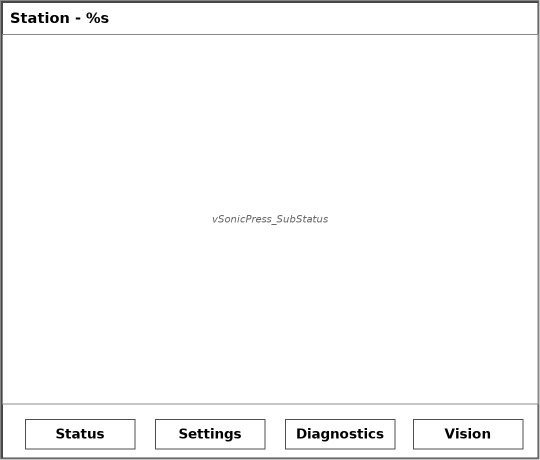
VISUALIZATION vSonicPress_Main  // 540x460
VAR_IN_OUT
	fbMachine: fbSonicPress;
	fbPIM: fbPIM_Station_V3;
	stTestParams:stSonicPress_TestParams;
END_VAR
    Rectangle (1,1 538x458)
    Rectangle (285,419 110x30), "Diagnostics"
        OnMouseClick: FrameSelectionChange Selection=SelectedFrame=57fd262e-2fea-4fde-aa72-b89d7183eaaf, Selection=2, GlobSel=AssignType=Expression, SelType=Locally
        OnMouseClick: execute { fbMachine.bTestMode:= FALSE; }
    Rectangle (155,419 110x30), "Settings"
        OnMouseClick: FrameSelectionChange Selection=SelectedFrame=57fd262e-2fea-4fde-aa72-b89d7183eaaf, Selection=1, GlobSel=AssignType=Expression, SelType=Locally
        OnMouseClick: execute { fbMachine.bTestMode:= FALSE; }
    Rectangle (25,419 110x30), "Status"
        OnMouseClick: FrameSelectionChange Selection=SelectedFrame=57fd262e-2fea-4fde-aa72-b89d7183eaaf, GlobSel=AssignType=Expression, SelType=Locally
    Frame (2,34 536x370)
        shows vSonicPress_SubStatus(fbMachine := fbMachine, fbPIM := fbPIM)
        shows vSonicPress_SubSettings(fbMachine := fbMachine, stTestParams := stTestParams)
        shows vSonicPress_SubDiag(fbMachine := fbMachine, fbPIM := fbPIM)
        shows vSonicPress_SubVision(fbMachine := fbMachine)
        p1079378287: stMachSettings
        p776352142: bVisuTestMode
    Rectangle (7,3 530x30), "Station - %s", text variable: fbPIM.sStationAlias
    Rectangle (413,419 110x30), "Vision", invisible if: NOT (fbPIM.sStationAlias='BS03PL01_1')
        OnMouseClick: FrameSelectionChange Selection=SelectedFrame=57fd262e-2fea-4fde-aa72-b89d7183eaaf, Selection=3, GlobSel=AssignType=Expression, SelType=Locally
END_VISUALIZATION

(* stored: Version 1.1.0.1, ProductVersion 3.1.4024.13
   Visu vSonicPress_Main: Id {3e7aea8e-4f5b-41d2-b069-a52afc41f3aa} *)
